Staubli VAL3: printScroll.pgx

program printScroll()
  local num i
  local num lX
  local num lY
begin
  //
  // put the scroll
  //
  if size(sItems)>nBottomY
    // find the percentage
    //windows style
    i=(size(sItems)-nBottomY+1)/(nFirst+1)
    // nokia style
    i=(size(sItems))/(nFirst+nView+1)
    lX=nTopX+nBottomX+1
    lY=roundUp((nBottomY)/i+nTopY)
    for i=nTopY+1 to nBottomY
      gotoxy(lX,i)
      if i==lY
        //
        put("■")
        //
      else
        put("│")
      endIf
    endFor
  endIf
end
